# EPICS substitutions: iocBoot/iocvirPV/DPU04.substitutions
file "../../db/virAi.template"{ pattern
{DPU,    num,    Temp}
{04,    0,    500}
{04,    1,    500}
{04,    2,    500}
{04,    3,    500}
{04,    4,    500}
{04,    5,    500}
{04,    6,    500}
{04,    7,    500}
{04,    8,    500}
{04,    9,    500}
{04,    10,    500}
{04,    11,    500}
{04,    12,    500}
{04,    13,    500}
{04,    14,    500}
{04,    15,    500}
{04,    16,    500}
{04,    17,    500}
{04,    18,    500}
{04,    19,    500}
{04,    20,    500}
{04,    21,    500}
{04,    22,    500}
{04,    23,    500}
{04,    24,    500}
{04,    25,    500}
{04,    26,    500}
{04,    27,    500}
{04,    28,    500}
{04,    29,    500}
{04,    30,    500}
{04,    31,    500}
{04,    32,    500}
{04,    33,    500}
{04,    34,    500}
{04,    35,    500}
{04,    36,    500}
{04,    37,    500}
{04,    38,    500}
{04,    39,    500}
{04,    40,    500}
{04,    41,    500}
{04,    42,    500}
{04,    43,    500}
{04,    44,    500}
{04,    45,    500}
{04,    46,    500}
{04,    47,    500}
{04,    48,    500}
{04,    49,    500}
{04,    50,    500}
{04,    51,    500}
{04,    52,    500}
{04,    53,    500}
{04,    54,    500}
{04,    55,    500}
{04,    56,    500}
{04,    57,    500}
{04,    58,    500}
{04,    59,    500}
{04,    60,    500}
{04,    61,    500}
{04,    62,    500}
{04,    63,    500}
{04,    64,    500}
{04,    65,    500}
{04,    66,    500}
{04,    67,    500}
{04,    68,    500}
{04,    69,    500}
{04,    70,    500}
{04,    71,    500}
{04,    72,    500}
{04,    73,    500}
{04,    74,    500}
{04,    75,    500}
{04,    76,    500}
{04,    77,    500}
{04,    78,    500}
{04,    79,    500}
{04,    80,    500}
{04,    81,    500}
{04,    82,    500}
{04,    83,    500}
{04,    84,    500}
{04,    85,    500}
{04,    86,    500}
{04,    87,    500}
{04,    88,    500}
{04,    89,    500}
{04,    90,    500}
{04,    91,    500}
{04,    92,    500}
{04,    93,    500}
{04,    94,    500}
{04,    95,    500}
{04,    96,    500}
{04,    97,    500}
{04,    98,    500}
{04,    99,    500}
{04,    100,    500}
{04,    101,    500}
{04,    102,    500}
{04,    103,    500}
{04,    104,    500}
{04,    105,    500}
{04,    106,    500}
{04,    107,    500}
{04,    108,    500}
{04,    109,    500}
{04,    110,    500}
{04,    111,    500}
{04,    112,    500}
{04,    113,    500}
{04,    114,    500}
{04,    115,    500}
{04,    116,    500}
{04,    117,    500}
{04,    118,    500}
{04,    119,    500}
{04,    120,    500}
{04,    121,    500}
{04,    122,    500}
{04,    123,    500}
{04,    124,    500}
{04,    125,    500}
{04,    126,    500}
{04,    127,    500}
{04,    128,    500}
{04,    129,    500}
{04,    130,    500}
{04,    131,    500}
{04,    132,    500}
{04,    133,    500}
{04,    134,    500}
{04,    135,    500}
{04,    136,    500}
{04,    137,    500}
{04,    138,    500}
{04,    139,    500}
{04,    140,    500}
{04,    141,    500}
{04,    142,    500}
{04,    143,    500}
{04,    144,    500}
{04,    145,    500}
{04,    146,    500}
{04,    147,    500}
{04,    148,    500}
{04,    149,    500}
{04,    150,    500}
{04,    151,    500}
{04,    152,    500}
{04,    153,    500}
{04,    154,    500}
{04,    155,    500}
{04,    156,    500}
{04,    157,    500}
{04,    158,    500}
{04,    159,    500}
{04,    160,    500}
{04,    161,    500}
{04,    162,    500}
{04,    163,    500}
{04,    164,    500}
{04,    165,    500}
{04,    166,    500}
{04,    167,    500}
{04,    168,    500}
{04,    169,    500}
{04,    170,    500}
{04,    171,    500}
{04,    172,    500}
{04,    173,    500}
{04,    174,    500}
{04,    175,    500}
{04,    176,    500}
{04,    177,    500}
{04,    178,    500}
{04,    179,    500}
{04,    180,    500}
{04,    181,    500}
{04,    182,    500}
{04,    183,    500}
{04,    184,    500}
{04,    185,    500}
{04,    186,    500}
{04,    187,    500}
{04,    188,    500}
{04,    189,    500}
{04,    190,    500}
{04,    191,    500}
{04,    192,    500}
{04,    193,    500}
{04,    194,    500}
{04,    195,    500}
{04,    196,    500}
{04,    197,    500}
{04,    198,    500}
{04,    199,    500}
}
